// Mitsubishi GX Works2 project: PLC 특수기능 (교번 출력, Flip-Flop)   PLC: Q03UDV

PROGRAM MAIN
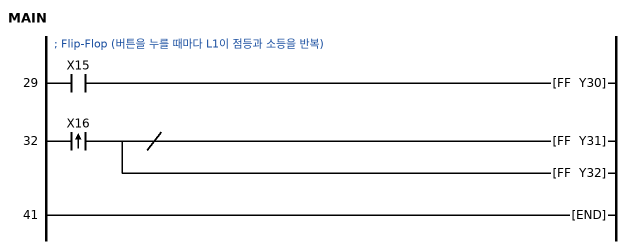
; Flip-Flop (버튼을 누를 때마다 L1이 점등과 소등을 반복)
29    LD      X15
      FF      Y30
32    LDP     X16
      MPS
      INV
      FF      Y31
      MPP
      FF      Y32
41    END
END_PROGRAM
